FUNCTION_BLOCK PUBLIC PAESensorBase EXTENDS PAModule
VAR_INPUT
END_VAR
VAR_OUTPUT
END_VAR
VAR
	_InputAddress : STRING;
	_SwitchingFrequency : DINT;
	_TotalAlarms : DINT;
END_VAR

METHOD FB_postinit
VAR_INPUT
	root : IACVariobatch;
END_VAR
SUPER^.FB_postinit(root);
root.OnPropertyChangedDInt(THIS^, 13, _SwitchingFrequency);
root.OnPropertyChangedDInt(THIS^, 14, _TotalAlarms);
root.OnPropertyChangedString(THIS^, 19, _InputAddress);
END_METHOD

{attribute 'monitoring' := 'call'}
//{attribute 'TcRpcEnable'}
PROPERTY PUBLIC InputAddress : STRING
GET // PUBLIC
InputAddress := _InputAddress;
END_GET
SET // PUBLIC
_InputAddress := InputAddress;
Root.OnPropertyChangedString(THIS^, 19, _InputAddress);
END_SET
END_PROPERTY

METHOD PUBLIC InvokeSetterString
VAR_INPUT
	PropertyID : INT;
	PropertyValue : STRING;
END_VAR
SUPER^.InvokeSetterString(PropertyID, PropertyValue);
IF PropertyID = 19 THEN
	InputAddress := PropertyValue;
END_IF
END_METHOD

METHOD OnInitMemory
VAR_INPUT
	root : IACVariobatch;
END_VAR
RegisterProperty(root, 13, GCL.cSizeDINT); // _SwitchingFrequency
RegisterProperty(root, 14, GCL.cSizeDINT); // _TotalAlarms
RegisterProperty(root, 19, GCL.cSizeSTRING); // InputAddress
SUPER^.OnInitMemory(root);
END_METHOD

{attribute 'monitoring' := 'call'}
//{attribute 'TcRpcEnable'}
PROPERTY PUBLIC SwitchingFrequency : DINT
GET
SwitchingFrequency := _SwitchingFrequency;
END_GET
SET
_SwitchingFrequency := SwitchingFrequency;
Root.OnPropertyChangedDInt(THIS^, 13, _SwitchingFrequency);
END_SET
END_PROPERTY

{attribute 'monitoring' := 'call'}
//{attribute 'TcRpcEnable'}
PROPERTY PUBLIC TotalAlarms : DINT
GET
TotalAlarms := _TotalAlarms;
END_GET
SET
_TotalAlarms := TotalAlarms;
Root.OnPropertyChangedDInt(THIS^, 14, _TotalAlarms);
END_SET
END_PROPERTY

END_FUNCTION_BLOCK

(* stored: Version 1.1.0.1, ProductVersion 3.1.4024.6
   POU PAESensorBase: Id {2dc5aea2-76a9-461c-85c2-a64f7833ddf5}, SpecialFunc None
   Method FB_postinit: Id {553449be-dad7-480b-9299-9061532627a5}
   Property InputAddress: Id {867c6579-09a3-4b24-9574-c2c54618edc1}
   Get Get: Id {4607d98b-ade6-458e-963e-009532d99776}
   Set Set: Id {0bf2c584-7a17-4de3-8b24-ca840e988d89}
   Method InvokeSetterString: Id {b6c2ef65-66b7-4541-bb15-d8bd1304478f}
   Method OnInitMemory: Id {b8cfcfc9-155f-4f95-a41a-f400427a7f82}
   Property SwitchingFrequency: Id {2224f919-5401-44a4-9805-42b6f0ba9168}
   Get Get: Id {4a61facb-0fb4-49bb-b98c-e59ca872aaf4}
   Set Set: Id {667c06d0-d5b1-4294-94cd-ff445f1253bc}
   Property TotalAlarms: Id {f38f6728-741f-4c58-aab7-e535e5e13065}
   Get Get: Id {a4264417-1b55-45f0-9b81-1ae3c9f767c8}
   Set Set: Id {7ded6128-ae59-4fc8-8d35-36e914c09094} *)
